FUNCTION_BLOCK FB_Visu_Pparam
VAR_IN_OUT
	stPParam_Visu:	ST_Param_Visu;
	stParamsUnsave:st_ParamsUnsave;
END_VAR
VAR
	nIdx:INT;
END_VAR

// LREAL


FOR nIdx:=1 TO cnParamsArrayLast BY 1 DO
	// Get
	stPParam_Visu.fLrealAktValue[nIdx]:=GetLreal(nVisuCount, nIdx);
	

	IF stPParam_Visu.bLrealSetValue[nIdx] THEN
		stPParam_Visu.bLrealSetValue[nIdx]:=FALSE;
		SetLreal(nVisuCount,nIdx, stPParam_Visu.fLrealNewValue[nidx]);
	END_IF
END_FOR

METHOD SetLreal : LREAL
VAR_INPUT
	nZone:	INT;
	nIdx:	INT;
	fValue:	LREAL;
END_VAR
VAR
END_VAR
CASE nIdx OF 
1:
	aaaPfwTempPparamFromHmi[nZone].Setpoint:=fValue;
2:
	aaaPfwTempPparamFromHmi[nZone].StandbySetpoint:=fValue;
3:
	aaaPfwTempPparamFromHmi[nZone].Setpoints[1]:=fValue;
4:
	aaaPfwTempPparamFromHmi[nZone].Setpoints[2]:=fValue;
5:
	aaaPfwTempPparamFromHmi[nZone].Setpoints[3]:=fValue;
6:
	aaaPfwTempPparamFromHmi[nZone].Setpoints[4]:=fValue;
7:
	aaaPfwTempPparamFromHmi[nZone].Setpoints[5]:=fValue;
8:
	aaaPfwTempPparamFromHmi[nZone].Threshold_PP:=fValue;
9:
	aaaPfwTempPparamFromHmi[nZone].Threshold_P:=fValue;
10:
	aaaPfwTempPparamFromHmi[nZone].Threshold_M:=fValue;
11:
	aaaPfwTempPparamFromHmi[nZone].Threshold_MM:=fValue;
12:
	aaaPfwTempPparamFromHmi[nZone].Openloop_Output:=fValue;
ELSE
	;
END_CASE

stParamsUnsave.pParams[nZone]:=TRUE;
END_METHOD

METHOD GetLreal : LREAL
VAR_INPUT
	nZone:	INT;
	nIdx:	INT;
END_VAR
VAR
END_VAR
CASE nIdx OF 
1:
	GetLreal:=aaaPfwTempPparamFromHmi[nZone].Setpoint;
2:
	GetLreal:=aaaPfwTempPparamFromHmi[nZone].StandbySetpoint;
3:
	GetLreal:=aaaPfwTempPparamFromHmi[nZone].Setpoints[1];
4:
	GetLreal:=aaaPfwTempPparamFromHmi[nZone].Setpoints[2];
5:
	GetLreal:=aaaPfwTempPparamFromHmi[nZone].Setpoints[3];
6:
	GetLreal:=aaaPfwTempPparamFromHmi[nZone].Setpoints[4];
7:
	GetLreal:=aaaPfwTempPparamFromHmi[nZone].Setpoints[5];
8:
	GetLreal:=aaaPfwTempPparamFromHmi[nZone].Threshold_PP;
9:
	GetLreal:=aaaPfwTempPparamFromHmi[nZone].Threshold_P;
10:
	GetLreal:=aaaPfwTempPparamFromHmi[nZone].Threshold_M;
11:
	GetLreal:=aaaPfwTempPparamFromHmi[nZone].Threshold_MM;
12:
	GetLreal:=aaaPfwTempPparamFromHmi[nZone].Openloop_Output;
	
ELSE
	GetLreal:=0.0;
END_CASE
END_METHOD

END_FUNCTION_BLOCK

(* stored: Version 1.1.0.1, ProductVersion 3.1.4018.5
   POU FB_Visu_Pparam: Id {2c87a0eb-457d-4781-87d1-1943a2914bff}, SpecialFunc None
   Method SetLreal: Id {0ebaa786-34c8-4f06-b779-2467b2b19035}
   Method GetLreal: Id {dae0f41a-8b0c-4b42-b11d-a6bae1b4878c} *)
